PROGRAM MAIN
VAR
	offSet AT %Q*:LREAL;
	cilindro:FB_CylinderSimul;
	avanca AT %I*: BOOL;
	recua AT %I*: BOOL;
	sensorFwd	AT %Q*: BOOL;
	sensorBwd	at %Q*: BOOL;
END_VAR

cilindro(
	moveFwd:=avanca , 
	moveBwd:= recua, 
	course:= 500, 
	moveVel:= 100, 
	cycleTime:= T#10MS, 
	sensorCylFwd=> sensorFwd, 
	sensorCylBwd=> sensorBwd, 
	currentPos=> , 
	posPercent=> offSet);

END_PROGRAM

(* stored: Version 1.1.0.1, ProductVersion 3.1.4024.12
   POU MAIN: Id {a74b5b65-3894-43db-b7be-7877929e6cee}, SpecialFunc None *)
